Universal Robots PolyScope program: mirror-me.urp

Program mirror-me (installation=mirror-me directory=/programs createdIn=3.2.19275 lastSavedIn=5.16.0 robotSerialNumber=20245201756)
Calibrated DH parameters: a=[0.000071, -0.502432, -0.570727, 0.000047, -0.000024, 0]; d=[0.180884, 276.390117, -282.568692, 6.352757, 0.119796, 0.115532]; alpha=[1.570625, -0.001266, 0.004349, 1.570389, -1.570248, 0]; deltaTheta=[0, -0.608501, 0.561455, 0.047042, -0.000001, 0]
InitVariablesNode variables(variable(name=mode, expression=0))
BeforeStart
  Script: write_output_boolean_register(64,  False )
  Wait Sleep waitTime=0.1
  mode := 0
  j := [0.,0,0,0,0,0]
Robot Program (runOnlyOnce=true)
  Script: write_output_boolean_register(64, False)
  Script: mode = read_input_integer_register(0)
  Loop While (checkContinuously=false) expression=mode < 3
    Loop While (checkContinuously=false) expression=mode ≟ 1
      MoveJ speed 15 deg/s, acceleration 40 deg/s^2 (useActiveTCP=true) feature=Base
        Waypoint Variable (Variable): variable(name=j)
      Script: write_output_boolean_register(64, True )
      Script: mode = read_input_integer_register(0)
      Script: sync()
    Loop While (checkContinuously=false) expression=(mode ≟ 2)
      Script: servoj(j, t=0.02, lookahead_time=0.5, gain=300)
      SuppressedNode
        Script: servoj(j)
      Script: mode = read_input_integer_register(0)
    Script: mode = read_input_integer_register(0)
    Script: write_output_boolean_register(64, False)
    Script: sync()
Thread Thread_1 (runOnlyOnce=false)
  Loop Forever
    tmp := [0,0,0,0,0,0]
    Script: tmp[0] = read_input_float_register(0)
    Script: tmp[1] = read_input_float_register(1)
    Script: tmp[2] = read_input_float_register(2)
    Script: tmp[3] = read_input_float_register(3)
    Script: tmp[4] = read_input_float_register(4)
    Script: tmp[5] = read_input_float_register(5)
    j := tmp
    Script: sync()
